FUNCTION_BLOCK FB_KF300 EXTENDS FB_Modbus_Tcp
(*
********************************************************************************
* Name: FB_KF300
*
* Author:  Automanh
* Version: 1.0.0
*
* Description:
*  KF300 Control for ShenChen
*
* Remarks:
*
* Revisions:
*   1.0 -AutomanH Rebuild
*********************************************************************************)
VAR_INPUT
	xIReset:BOOL;
	xIManualMode:BOOL;
	xIAutoMode:BOOL;
	xIEstop:BOOL;
	xIDeviceRunning:BOOL;
	LocalClient:stModbusPara;
	stRunPara	:ST_SetPara;//运行参数	
	stDeviceOpe	: stEasyPumpHmi;//操作按钮
END_VAR
VAR_OUTPUT
 	xQRdyCmd:BOOL;
	xQError:BOOL;
	xQBusy:BOOL;
	xQDone:BOOL;
	strQErrorID:STRING;
	xQCalibrationOK:BOOL;
	rMaxRunTime	:REAL;//最大运行时间,单位s
	rMinRunTime	:REAL;//最小运行时间,单位s
END_VAR
VAR
 	xStart:BOOL;
 {attribute 'tc_no_symbol'}
 iParaStep,iOldParaStep,iRunStep,iOldRunStep:INT;
 {attribute 'tc_no_symbol'}
 iCalibStep,iOldCalibStep:INT;
 {attribute 'tc_no_symbol'}
 stLocalPara:ST_LocalPara;
 {attribute 'tc_no_symbol'}
 stPara,stRun,stCalibInit,stCalibAction,stAdjust:ST_StepStatus; 
 {attribute 'tc_no_symbol'}
 stPump:st_EasyPump;
  {attribute 'tc_no_symbol'}
	tTimeout:ARRAY[1..5] OF TON;
 {attribute 'tc_no_symbol'}
	// 蠕动泵读取的液量
	rCurrVolum: REAL;
	{attribute 'tc_no_symbol'}
	//从蠕动泵读取的参数
	stReadPara:ST_ReadPara;
	{attribute 'tc_no_symbol'}
	// 数据数组
	arwData: ARRAY[1..2] OF WORD;
	{attribute 'tc_no_symbol'}
	eErrorID		: PumpError;(*错误码*)
	{attribute 'tc_no_symbol'}
	// 根据设定计算的转速
	rSetSpeed: REAL;
	{attribute 'tc_no_symbol'}
	// 设定的数据
	arwSetData: ARRAY [1..2] OF WORD;
	{attribute 'tc_no_symbol'}
	// 虚拟的较大时间
	rVirtualTime: REAL;
	{attribute 'tc_no_symbol'}
	OperR_TRIG:ARRAY[1..20] OF R_TRIG;
	{attribute 'tc_no_symbol'}
	// 循环计数
	i: INT;
	{attribute 'tc_no_symbol'}
	// 操作类型
	iOperType: INT;
	{attribute 'tc_no_symbol'}
	iOperCounter:INT;
	{attribute 'tc_no_symbol'}
	artDelay:ARRAY[1..5] OF TON;
	{attribute 'tc_no_symbol'}
	tSetTime:TIME;
	tModuleDelay:TON;
	iCalibNum:INT:=1;//校准灌装次数
END_VAR

MEMCPY(ADR(SUPER^.stModbusPara),ADR(LocalClient),SIZEOF(localClient));
SUPER^.M_Modbus();
ACT_RunPara();
ACT_Operation();
ACT_Running();
ACT_ParaCalc();
ACT_Calibration();
ACT_Reset();
ACT_Error();

ACTION ACT_Calibration:
CASE iCalibStep OF
 			0://等待启动
				 IF	stCalibInit.xStart THEN
							stCalibInit.xStart:=FALSE;
							stCalibInit.xBusy:=TRUE;
							stCalibInit.xDone:=FALSE;	
							iCalibStep:=10;//初始化校准参数
				 ELSIF stCalibAction.xStart THEN
						 	 stCalibAction.xStart :=FALSE;
							 stCalibAction.xBusy :=TRUE;
							 stCalibAction.xDone :=FALSE;
							 iCalibStep:=20;//校准
					ELSIF stAdjust.xStart THEN
					 		 stAdjust.xStart :=FALSE;
							 stAdjust.xBusy :=TRUE;
							 stAdjust.xDone :=FALSE;
							 iCalibStep:=30;//微调
				 END_IF
			10://初始化校准参数
					 iOldCalibStep:=iCalibStep;
					 arwDataWriteRegs[1]:=1;
					 wQuantityWriteRegs:=1;
					 wMBAddWriteRegs:=2007;
					 xWriteRegs:=TRUE;
					 IF  fbWriteRegs.bBusy THEN
							 xWriteRegs:=FALSE;
							 iCalibStep:=iCalibStep+1;
					END_IF
			11://液量设定完成
							 iOldCalibStep:=iCalibStep;
						 IF  NOT 	fbWriteRegs.bBusy AND  NOT  	fbWriteRegs.bError THEN
										iCalibStep:=iCalibStep+1;
							ELSIF   	fbReadRegs.bError THEN
									 iCalibStep:=999;				
									 eErrorID:=PumpError.FLT_SET_PARA;					
							END_IF		
		
			12://初始化校准参数完成
						 stCalibInit.xBusy:=FALSE;
							stCalibInit.xDone:=TRUE;	
						 	iCalibStep:=0;
						 
			
			 20://检查实际液量与设定液量的误差范围
					 IF   (stLocalPara.rFluVolumeSet - stLocalPara.iModuleRealVolume )<stLocalPara.rFluVolumeSet*0.5 THEN
							 //误差不能超过0.3ml
							 iCalibStep:=iCalibStep +1;				
					 ELSE
								 eERRORID := PumpError.FLT_Calib_OverFlow;//误差过大
								 iCalibStep:=999;	
					 END_IF
			 21://需要设定实际液量--实际液量最好是三组液量的平均值
							iOldCalibStep:=iCalibStep;
							MEMCPY(ADR(arwSetData[1]),ADR(stLocalPara.iModuleRealVolume),SIZEOF(stLocalPara.iModuleRealVolume) ); 
							arwDataWriteRegs[1]:=arwSetData[2];
							arwDataWriteRegs[2]:=arwSetData[1];
							wQuantityWriteRegs:=2;
							wMBAddWriteRegs:=2004;
							xWriteRegs:=TRUE;
							IF  fbWriteRegs.bBusy THEN
									xWriteRegs:=FALSE;
									 iCalibStep:=iCalibStep +1;		
						 END_IF
			 22://液量设定完成
							iOldCalibStep:=iCalibStep;
						 IF  NOT 	fbWriteRegs.bBusy AND  NOT  	fbWriteRegs.bError THEN
											 iCalibStep:=iCalibStep +1;		
							ELSIF   	fbReadRegs.bError THEN
										 iCalibStep:=999;				
										 eErrorID:=PumpError.FLT_CALIB_PARA;					
							END_IF		
			 23://校准实际液量设定结束
						 stCalibAction.xBusy :=FALSE;
						 stCalibAction.xDone :=TRUE;
						 iCalibStep:=0;				 
			30://校准微调-微调幅度为(设定量*0.001),这里要根据客户要求的精度进行调整
					 xQCalibrationOK:=FALSE;
					 iCalibStep:=iCalibStep +1;
			31://检测数据是否在精度范围内
					 iOldCalibStep:=iCalibStep;
					 IF  stLocalPara.iModuleRealVolume>=stLocalPara.rFluVolumeSet-(stLocalPara.rFluVolumeSet*stLocalPara.iAccuracySet) AND 
							 stLocalPara.iModuleRealVolume<=stLocalPara.rFluVolumeSet+(stLocalPara.rFluVolumeSet*stLocalPara.iAccuracySet) THEN
							 	 xQCalibrationOK:=TRUE;
								 iCalibStep:=36;
					ELSIF stLocalPara.iModuleRealVolume>=stLocalPara.rFluVolumeSet-(stLocalPara.rFluVolumeSet*stLocalPara.iAccuracySet) THEN
								 iCalibStep:=iCalibStep +1;	//需要减小
					ELSIF  stLocalPara.iModuleRealVolume<=stLocalPara.rFluVolumeSet+(stLocalPara.rFluVolumeSet*stLocalPara.iAccuracySet) THEN
								 iCalibStep:=iCalibStep +3;	//需要增大
					END_IF
			32://发送微调指令
					iOldParaStep:=iParaStep;
					arwDataWriteRegs[1]:=0;
					wQuantityWriteRegs:=1;
					wMBAddWriteRegs:=2006;
					xWriteRegs:=TRUE;
					IF  fbWriteRegs.bBusy THEN
							xWriteRegs:=FALSE;
							iCalibStep:=iCalibStep+1;
				 END_IF
		  33://微调执行完成
					 iOldParaStep:=iParaStep;
					 IF  NOT 	fbWriteRegs.bBusy AND  NOT  	fbWriteRegs.bError THEN
									 iCalibStep:=36;
						ELSIF   	fbReadRegs.bError THEN
								 iCalibStep:=999;				
								 eErrorID:=PumpError.FLT_SET_PARA;					
						END_IF			 
			34://发送微调指令
					iOldParaStep:=iParaStep;
					arwDataWriteRegs[1]:=1;
					wQuantityWriteRegs:=1;
					wMBAddWriteRegs:=2006;
					xWriteRegs:=TRUE;
					IF  fbWriteRegs.bBusy THEN
							xWriteRegs:=FALSE;
							iCalibStep:=iCalibStep+1;
				 END_IF
		  35://微调执行完成
					 iOldParaStep:=iParaStep;
					 IF  NOT 	fbWriteRegs.bBusy AND  NOT  	fbWriteRegs.bError THEN
									 iCalibStep:=36;
						ELSIF   	fbReadRegs.bError THEN
								 iCalibStep:=999;				
								 eErrorID:=PumpError.FLT_SET_PARA;					
						END_IF			 			
			 36://微调完成
							 stAdjust.xBusy :=FALSE;
							 stAdjust.xDone :=TRUE;
							 iCalibStep:=0;//校准			
END_CASE
 //防止程序二次执行
 IF	stCalibInit.xBusy THEN
			stCalibInit.xStart:=FALSE;
 ELSIF stCalibAction.xBusy THEN
			stCalibAction.xStart :=FALSE;
 ELSIF stAdjust.xBusy THEN
			stAdjust.xStart :=FALSE;
 END_IF
END_ACTION

ACTION ACT_Error:
tTimeout[1](IN:= iParaStep =iOldParaStep AND iParaStep<>0 , PT:= T#15S, Q=> , ET=> );
tTimeout[2](IN:= iRunStep =iOldRunStep AND iRunStep<>0 , PT:= T#15S, Q=> , ET=> );
tTimeout[3](IN:= iCalibStep =iOldCalibStep AND iCalibStep<>0 , PT:= T#15S, Q=> , ET=> );
IF		tTimeout[1].Q THEN
	  	stPara.xError:=TRUE;
	  	stPara.xBusy:=FALSE;
			eErrorID:=PumpError.FLT_CMD_TIMEOUT;
	    iParaStep := 999;
END_IF

IF		tTimeout[2].Q THEN
			stRun.xError:=TRUE;
			stRun.xBusy:=FALSE;
			eErrorID:=PumpError.FLT_CMD_TIMEOUT;
			iRunStep := 999;
END_IF

IF		tTimeout[3].Q THEN
			stAdjust.xError:=TRUE;
			stAdjust.xBusy:=FALSE;
			eErrorID:=PumpError.FLT_CMD_TIMEOUT;
			iCalibStep := 999;
END_IF

IF  eErrorID <> PumpError.NO_ERROR THEN
		xQError:=TRUE;
END_IF
//报错内容输出
CASE eErrorID OF 
		 PumpError.No_ERROR:
			 strQErrorID:='NO ERROR';
		 PumpError.FLT_PARA:
			 strQErrorID:='FLT_PARA';
		 PumpError.FLT_FLUVOLUM_TIME_PARA:
			 strQErrorID:='FLT_FLUVOLUM_TIME_PARA';
		 PumpError.FLT_SET_PARA:
			 strQErrorID:='FLT_SET_PARA';	
		 PumpError.FLT_CMD_TIMEOUT:
			 strQErrorID:='FLT_CMD_TIMEOUT';	
		 PumpError.FLT_RUN_ERROR:
			 strQErrorID:='FLT_RUN_ERROR';
		 PumpError.FLT_Calib_OverFlow:
			 strQErrorID:='FLT_Calib_OverFlow';	
		 PumpError.FLT_CALIB_PARA:
			 strQErrorID:='FLT_CALIB_PARA';		
		 PumpError.FLT_CONFIGURE_PARA:
			 strQErrorID:='FLT_CONFIGURE_PARA';		
END_CASE
END_ACTION

ACTION ACT_Operation:
OperR_TRIG[1](CLK:= (xIManualMode AND  stDeviceOpe.xPush_Hmi[1]) OR((xIAutoMode OR  xIDeviceRunning) AND stDeviceOpe.xPush_Auto[1]) , Q=> );	//Push
OperR_TRIG[2](CLK:= (xIManualMode AND  stDeviceOpe.xPush_Hmi[2]) OR((xIAutoMode OR  xIDeviceRunning) AND stDeviceOpe.xPush_Auto[2]) , Q=> );	//Push
OperR_TRIG[3](CLK:= (xIManualMode AND  stDeviceOpe.xPush_Hmi[3]) OR((xIAutoMode OR  xIDeviceRunning) AND stDeviceOpe.xPush_Auto[3]) , Q=> );	//Push
OperR_TRIG[4](CLK:= (xIManualMode AND  stDeviceOpe.xPush_Hmi[4]) OR((xIAutoMode OR  xIDeviceRunning) AND stDeviceOpe.xPush_Auto[4]) , Q=> );	//Push
OperR_TRIG[5](CLK:= (xIManualMode AND  stDeviceOpe.xPush_Hmi[5]) OR((xIAutoMode OR  xIDeviceRunning) AND stDeviceOpe.xPush_Auto[5]) , Q=> );	//Push
OperR_TRIG[6](CLK:= (xIManualMode AND  stDeviceOpe.xPull_Hmi[1]) OR((xIAutoMode OR  xIDeviceRunning) AND stDeviceOpe.xPull_Auto[1]) , Q=> );	//Pull
OperR_TRIG[7](CLK:= (xIManualMode AND  stDeviceOpe.xPull_Hmi[2]) OR((xIAutoMode OR  xIDeviceRunning) AND stDeviceOpe.xPull_Auto[2]) , Q=> );	//Pull
OperR_TRIG[8](CLK:= (xIManualMode AND  stDeviceOpe.xPull_Hmi[3]) OR((xIAutoMode OR  xIDeviceRunning) AND stDeviceOpe.xPull_Auto[3]) , Q=> );	//Pull
OperR_TRIG[9](CLK:= (xIManualMode AND  stDeviceOpe.xPull_Hmi[4]) OR((xIAutoMode OR  xIDeviceRunning) AND stDeviceOpe.xPull_Auto[4]) , Q=> );	//Pull
OperR_TRIG[10](CLK:= (xIManualMode AND  stDeviceOpe.xPull_Hmi[5]) OR((xIAutoMode OR  xIDeviceRunning) AND stDeviceOpe.xPull_Auto[5]) , Q=> );	//Pull
OperR_TRIG[11](CLK:= (xIManualMode AND  stDeviceOpe.xModulePush_Hmi) OR((xIAutoMode OR  xIDeviceRunning) AND stDeviceOpe.xModulePush_Auto) , Q=> );		//ModulePush	
OperR_TRIG[12](CLK:= (xIManualMode AND  stDeviceOpe.xFullSpeedPush_Hmi) OR((xIAutoMode OR  xIDeviceRunning) AND stDeviceOpe.xFullSpeedPush_Auto) , Q=> );//FullSpeedPush
OperR_TRIG[13](CLK:= (xIManualMode AND  stDeviceOpe.xFullSpeedPull_Hmi) OR((xIAutoMode OR  xIDeviceRunning) AND stDeviceOpe.xFullSpeedPull_Auto) , Q=> );//FullSpeedPull
OperR_TRIG[14](CLK:= (xIManualMode AND  stDeviceOpe.xFullSpeedStop_Hmi) OR((xIAutoMode OR  xIDeviceRunning) AND stDeviceOpe.xFullSpeedStop_Auto) , Q=> );//FullSpeedStop
OperR_TRIG[15](CLK:= (xIManualMode AND  stDeviceOpe.xStop_Hmi) OR((xIAutoMode OR  xIDeviceRunning) AND stDeviceOpe.xStop_Auto  ) , Q=> );//Stop
OperR_TRIG[16](CLK:= (xIManualMode AND  stDeviceOpe.xCalibAction_Hmi) OR((xIAutoMode OR  xIDeviceRunning) AND stDeviceOpe.xCalibAction_Auto) , Q=> );//Calibration Action
OperR_TRIG[17](CLK:= (xIManualMode AND  stDeviceOpe.xCalibInit_Hmi) OR((xIAutoMode OR  xIDeviceRunning) AND stDeviceOpe.xCalibInit_Auto), Q=> );//Calibration Init
OperR_TRIG[18](CLK:= (xIManualMode AND  stDeviceOpe.xAdjust_Hmi) OR((xIAutoMode OR  xIDeviceRunning) AND stDeviceOpe.xAdjust_Auto), Q=> );//Adjust
OperR_TRIG[19](CLK:= xIEstop, Q=> );//Estop

FOR  i:= 1 TO 20 BY 1 DO
 	IF   OperR_TRIG[i].Q THEN
				iOperCounter:= i;
				xStart:=TRUE;
				EXIT;
	END_IF
END_FOR
//Push
FOR  i:=1 TO 5 BY 1 DO
 		IF   iOperCounter =i THEN
		 		stLocalPara.rFluVolumeSet	:=stRunPara.rPushFluVolume[i];
				stLocalPara.rRuntimeSet	:=stRunPara.rPushRuntime[i];
				stLocalPara.iCycleNumber	:=stRunPara.iPushCycleNumber[i];
				stLocalPara.iBackAngle:=stRunPara.iPushBackAngle[i];
				stLocalPara.iDirectionSet:=stRunPara.iDirectionSet;
				stLocalPara.rVirualTime:=rMaxRunTime -1;
				iOperType:=stOperType.iPush;
		END_IF
END_FOR
//pull
FOR  i:=6 TO 10 BY 1 DO
 		IF   iOperCounter =i THEN
		 		stLocalPara.rFluVolumeSet	:=stRunPara.rPullFluVolume[i-5];
				stLocalPara.rRuntimeSet	:=stRunPara.rPullRuntime[i-5];
				stLocalPara.iCycleNumber	:=stRunPara.iPullCycleNumber[i-5];
				stLocalPara.iBackAngle:=stRunPara.iPullBackAngle[i-5];
				stLocalPara.iDirectionSet:=ABS(1-stRunPara.iDirectionSet);
				stLocalPara.rVirualTime:=rMaxRunTime -1;
				iOperType:=stOperType.iPull;
		END_IF
END_FOR 
 //Module Push
IF   iOperCounter =11 THEN
		 		stLocalPara.rFluVolumeSet	:=stRunPara.rCalFluVolume;
				stLocalPara.rRuntimeSet	 :=stRunPara.rCalTime;
				stLocalPara.iCycleNumber :=stRunPara.rCalNum;
				stLocalPara.iBackAngle:=stRunPara.rCalBackAngle;
				stLocalPara.iDirectionSet:=stRunPara.iDirectionSet;
				stLocalPara.iModuleAdress:=stRunPara.iModuleAdress;
				stLocalPara.iModuleSpeed:= stRunPara.rCalFluVolume * 60.0/(stRunPara.rSpeedRatio* stRunPara.rCalTime);
				stLocalPara.rVirualTime:=rMaxRunTime -1;
				iOperType:=stOperType.iModulePush;
////FullSpeedPush
ELSIF  iOperCounter =12 THEN
 				stLocalPara.iDirectionSet:=stRunPara.iDirectionSet;
 				iOperType:=stOperType.iFullSpeedPush;
ELSIF  iOperCounter =13 THEN
 			stLocalPara.iDirectionSet:=ABS(1-stRunPara.iDirectionSet);
 			iOperType:=stOperType.iFullSpeedPull;
ELSIF  iOperCounter =14 THEN
 			iOperType:=stOperType.iFullSpeedStop;
ELSIF  iOperCounter =15 OR iOperCounter =19  THEN
 			iOperType:=stOperType.iStop;
ELSIF  iOperCounter =16  THEN//Calibration
 			stLocalPara.iModuleRealVolume:=stRunPara.rModuleRealFluVolume;
 			iOperType:=stOperType.iCalibAction;
ELSIF  iOperCounter =17  THEN
 			iOperType:=stOperType.iCalibInit;	
ELSIF    iOperCounter =18 THEN //adjust
 			stLocalPara.iModuleRealVolume:=stRunPara.rModuleRealFluVolume;
 			stLocalPara.iAccuracySet:=stRunPara.iAccuracySet;
 			iOperType:=stOperType.iAdjust;	
END_IF


MEMSET(ADR(stDeviceOpe),0,SIZEOF(stDeviceOpe));
END_ACTION

ACTION ACT_ParaCalc:
//
(*************************检测配置参数是否匹配成功*********************************)
IF stRunPara.iPumpType=RudongPump_PumpType.DFPluse THEN
	//MiniPump泵头
	IF  stRunPara.iPumpTypeSet=RudongPump_PumpHeadType.MiniPump01 THEN
		stPump.iPumpType:=0;//泵头值为0
			IF stRunPara.iHosePipeTypeSet=RudongPump_SoftPipeType.P13 THEN//13#软管
				stPump.iHosePipeType:=13;//软管类型值13
				IF  stLocalPara.rFluVolumeSet*1000/135<0.1 THEN
					rMaxRunTime:=	0.1;
				ELSE
					rMaxRunTime:=	stLocalPara.rFluVolumeSet*1000/135;
				END_IF
				rMaxRunTime:=	(stLocalPara.rFluVolumeSet/0.45)*0.2;//最大流量(0.45微升/秒,0.0024ml/min)	
			ELSIF stRunPara.iHosePipeTypeSet=RudongPump_SoftPipeType.P14 THEN//14#软管
					stPump.iHosePipeType:=13;//软管类型值13
				IF stLocalPara.rFluVolumeSet*1000/570<0.1 THEN
							rMinRunTime:=	0.1;
				ELSE
						rMinRunTime:=	stLocalPara.rFluVolumeSet*1000/135;
				END_IF
				rMaxRunTime:=	(stLocalPara.rFluVolumeSet/1.9)*0.2;	
			ELSIF stRunPara.iHosePipeTypeSet=RudongPump_SoftPipeType.P19 THEN//19#软管
				stPump.iHosePipeType:=19;
				IF stLocalPara.rFluVolumeSet*1000/1240<0.1 THEN
					rMinRunTime:=	0.1;
				ELSE
					rMinRunTime:=	stLocalPara.rFluVolumeSet*1000/1240;
				END_IF
					rMaxRunTime:=	(stLocalPara.rFluVolumeSet*1000/4.13)*0.2;		
			ELSIF stRunPara.iHosePipeTypeSet=RudongPump_SoftPipeType.P16 THEN//16#软管
					stPump.iHosePipeType:=16;
				IF stLocalPara.rFluVolumeSet*1000/1880<0.1 THEN
					rMinRunTime:=	0.1;
				ELSE
					rMinRunTime:=	stLocalPara.rFluVolumeSet*1000/1880;
				END_IF
				rMaxRunTime:=	(stLocalPara.rFluVolumeSet*1000/6.28)*0.2;	
			ELSIF stRunPara.iHosePipeTypeSet=RudongPump_SoftPipeType.P25 THEN//25#软管
					stPump.iHosePipeType:=25;
				IF stLocalPara.rFluVolumeSet*1000/3100<0.1 THEN
					rMinRunTime:=	0.1;
				ELSE
					rMinRunTime:=	stLocalPara.rFluVolumeSet*1000/3100;
				END_IF
				rMaxRunTime:=	(stLocalPara.rFluVolumeSet*1000/10.33)*0.2;			
		ELSE
				eERRORID:=RudongPump_ERROR.FLT_CONFIGURE_PARA;		
		END_IF
	//UD15
	ELSIF  stRunPara.iPumpTypeSet=RudongPump_PumpHeadType.UD15 THEN
				stPump.iHosePipeType:=1;//泵头值为0
			IF stRunPara.iHosePipeTypeSet=RudongPump_SoftPipeType.P16 THEN//16#软管
				stPump.iHosePipeType:=16;
				IF stLocalPara.rFluVolumeSet*1000/4000<0.1 THEN
					rMinRunTime:=	0.1;
				ELSE
					rMinRunTime:=	stLocalPara.rFluVolumeSet*1000/4000;
				END_IF
				rMaxRunTime:=	(stLocalPara.rFluVolumeSet*1000/13.33)*0.2;		
			ELSIF stRunPara.iHosePipeTypeSet=RudongPump_SoftPipeType.P17 THEN//17#软管
				stPump.iHosePipeType:=17;
				IF stLocalPara.rFluVolumeSet*1000/15000<0.1 THEN
					rMinRunTime:=	0.1;
				ELSE
					rMinRunTime:=	stLocalPara.rFluVolumeSet*1000/15000;
				END_IF
				rMaxRunTime:=	(stLocalPara.rFluVolumeSet*1000/50)*0.2;	
			ELSIF stRunPara.iHosePipeTypeSet=RudongPump_SoftPipeType.P25 THEN//25#软管
				stPump.iHosePipeType:=25;
				IF stLocalPara.rFluVolumeSet*1000/8000<0.1 THEN
					rMinRunTime:=	0.1;
				ELSE
					rMinRunTime:=	stLocalPara.rFluVolumeSet*1000/8000;
				END_IF
				 rMaxRunTime:=	(stLocalPara.rFluVolumeSet*1000/26.66)*0.2;			
		ELSE
				eERRORID:=RudongPump_ERROR.FLT_CONFIGURE_PARA;		
		END_IF
	//HandyPump01泵头
ELSIF  stRunPara.iPumpTypeSet=RudongPump_PumpHeadType.HandyPump01 THEN
 			IF stRunPara.iHosePipeTypeSet=RudongPump_SoftPipeType.P13 THEN//13#软管,三滚轮
				IF stLocalPara.rFluVolumeSet*1000/155<0.1 THEN
					rMinRunTime:=	0.1;
				ELSE
					rMinRunTime:=	stLocalPara.rFluVolumeSet*1000/155;
				END_IF
					rMaxRunTime:=	(stLocalPara.rFluVolumeSet*1000/0.51)*0.2;	
		
	(*	IF stRunPara.iHosePipeTypeSet=RudongPump_SoftPipeType.P13 THEN//13#软管,三滚轮
			iMinRunTime:=	(rFluVolumeSet/10)*60;
			iMaxRunTime:=	(rFluVolumeSet/0.0033)*60;	
		ELSIF stRunPara.iHosePipeTypeSet=RudongPump_SoftPipeType.P14 THEN//14#软管,三滚轮
			iMinRunTime:=	(rFluVolumeSet/56)*60;
			iMaxRunTime:=	(rFluVolumeSet/0.0187)*60;		
		ELSIF stRunPara.iHosePipeTypeSet=RudongPump_SoftPipeType.P19 THEN//19#软管,三滚轮
			iMinRunTime:=	(rFluVolumeSet/111)*60;
			iMaxRunTime:=	(rFluVolumeSet/0.0371)*60;
		ELSIF stRunPara.iHosePipeTypeSet=RudongPump_SoftPipeType.P16 THEN//16#软管,三滚轮
			iMinRunTime:=	(rFluVolumeSet/190)*60;
			iMaxRunTime:=	(rFluVolumeSet/0.0636)*60;		
		ELSIF stRunPara.iHosePipeTypeSet=RudongPump_SoftPipeType.P25 THEN//25#软管,三滚轮
			iMinRunTime:=	(rFluVolumeSet/365)*60;
			iMaxRunTime:=	(rFluVolumeSet/0.1219)*60;
	*)
		ELSE
				eERRORID:=RudongPump_ERROR.FLT_CONFIGURE_PARA;						
		END_IF
	END_IF
ELSE
		eERRORID:=RudongPump_ERROR.FLT_CONFIGURE_PARA;
END_IF


(*
//MiniPump01泵头
IF  stRunPara.iPumpTypeSet=RudongPump_PumpHeadType.MiniPump01 THEN
		IF stRunPara.iHosePipeTypeSet=RudongPump_SoftPipeType.P13 THEN//13#软管
			iMinRunTime:=	(rFluVolumeSet/8)*60;//最大流量(135微升/秒,8.28ml/min)
			iMaxRunTime:=	(rFluVolumeSet/0.45)*60;//最大流量(0.45微升/秒,0.0024ml/min)	
		ELSIF stRunPara.iHosePipeTypeSet=RudongPump_SoftPipeType.P14 THEN//14#软管
			iMinRunTime:=	(rFluVolumeSet/33)*60;
			iMaxRunTime:=	(rFluVolumeSet/1.9)*60;
		ELSIF stRunPara.iHosePipeTypeSet=RudongPump_SoftPipeType.P19 THEN//19#软管
			iMinRunTime:=	(rFluVolumeSet/77)*60;
			iMaxRunTime:=	(rFluVolumeSet/4.13)*60;	
		ELSIF stRunPara.iHosePipeTypeSet=RudongPump_SoftPipeType.P16 THEN//16#软管
			iMinRunTime:=	(rFluVolumeSet/114)*60;
			iMaxRunTime:=	(rFluVolumeSet/6.28)*60;	
		ELSIF stRunPara.iHosePipeTypeSet=RudongPump_SoftPipeType.P25 THEN//25#软管
			iMinRunTime:=	(rFluVolumeSet/190)*60;
			iMaxRunTime:=	(rFluVolumeSet/10.33)*60;		
		ELSIF stRunPara.iHosePipeTypeSet=RudongPump_SoftPipeType.P1_1 THEN//1x1#软管
			iMinRunTime:=	(rFluVolumeSet/15)*60;
			iMaxRunTime:=	(rFluVolumeSet/4.5)*60;	
		ELSIF stRunPara.iHosePipeTypeSet=RudongPump_SoftPipeType.P2_1 THEN//2x1#软管
			iMinRunTime:=	(rFluVolumeSet/54)*60;
			iMaxRunTime:=	(rFluVolumeSet/4.5)*60;		
		ELSIF stRunPara.iHosePipeTypeSet=RudongPump_SoftPipeType.P2_5_1 THEN//2.5x1#软管
			iMinRunTime:=	(rFluVolumeSet/76)*60;
			iMaxRunTime:=	(rFluVolumeSet/5)*60;		
		ELSIF stRunPara.iHosePipeTypeSet=RudongPump_SoftPipeType.P3_1 THEN//3x1#软管
			iMinRunTime:=	(rFluVolumeSet/108)*60;
			iMaxRunTime:=	(rFluVolumeSet/5)*60;
	ELSE
			eERRORID:=RudongPump_ERROR.FLT_CONFIGURE_PARA;		
	END_IF		
	
//MiniPump02泵头
ELSIF  stRunPara.iPumpTypeSet=RudongPump_PumpHeadType.MiniPump02 THEN
	IF stRunPara.iHosePipeTypeSet=RudongPump_SoftPipeType.P1_1 THEN//1x1#软管
		iMinRunTime:=	(rFluVolumeSet/15.01)*60;
		iMaxRunTime:=	(rFluVolumeSet/0.005)*60;	
	ELSIF stRunPara.iHosePipeTypeSet=RudongPump_SoftPipeType.P2_1 THEN//2x1#软管
		iMinRunTime:=	(rFluVolumeSet/54.63)*60;
		iMaxRunTime:=	(rFluVolumeSet/0.018)*60;		
	ELSIF stRunPara.iHosePipeTypeSet=RudongPump_SoftPipeType.P2_5_1 THEN//2.5x1#软管
		iMinRunTime:=	(rFluVolumeSet/76.84)*60;
		iMaxRunTime:=	(rFluVolumeSet/0.0256)*60;
	ELSE
			eERRORID:=RudongPump_ERROR.FLT_CONFIGURE_PARA;						
	END_IF	

//HandyPump01泵头
ELSIF  stRunPara.iPumpTypeSet=RudongPump_PumpHeadType.HandyPump01 THEN
	IF stRunPara.iHosePipeTypeSet=RudongPump_SoftPipeType.P13 THEN//13#软管,三滚轮
		iMinRunTime:=	(rFluVolumeSet/10)*60;
		iMaxRunTime:=	(rFluVolumeSet/0.0033)*60;	
	ELSIF stRunPara.iHosePipeTypeSet=RudongPump_SoftPipeType.P14 THEN//14#软管,三滚轮
		iMinRunTime:=	(rFluVolumeSet/56)*60;
		iMaxRunTime:=	(rFluVolumeSet/0.0187)*60;		
	ELSIF stRunPara.iHosePipeTypeSet=RudongPump_SoftPipeType.P19 THEN//19#软管,三滚轮
		iMinRunTime:=	(rFluVolumeSet/111)*60;
		iMaxRunTime:=	(rFluVolumeSet/0.0371)*60;
	ELSIF stRunPara.iHosePipeTypeSet=RudongPump_SoftPipeType.P16 THEN//16#软管,三滚轮
		iMinRunTime:=	(rFluVolumeSet/190)*60;
		iMaxRunTime:=	(rFluVolumeSet/0.0636)*60;		
	ELSIF stRunPara.iHosePipeTypeSet=RudongPump_SoftPipeType.P25 THEN//25#软管,三滚轮
		iMinRunTime:=	(rFluVolumeSet/365)*60;
		iMaxRunTime:=	(rFluVolumeSet/0.1219)*60;
	ELSE
			eERRORID:=RudongPump_ERROR.FLT_CONFIGURE_PARA;						
	END_IF

//HandyPump02泵头
ELSIF  stRunPara.iPumpTypeSet=RudongPump_PumpHeadType.HandyPump02 THEN
	IF stRunPara.iHosePipeTypeSet=RudongPump_SoftPipeType.P13 THEN//13#软管,三滚轮
		iMinRunTime:=	(rFluVolumeSet/10)*60;
		iMaxRunTime:=	(rFluVolumeSet/0.0033)*60;	
	ELSIF stRunPara.iHosePipeTypeSet=RudongPump_SoftPipeType.P14 THEN//14#软管,三滚轮
		iMinRunTime:=	(rFluVolumeSet/56)*60;
		iMaxRunTime:=	(rFluVolumeSet/0.0187)*60;		
	ELSIF stRunPara.iHosePipeTypeSet=RudongPump_SoftPipeType.P19 THEN//19#软管,三滚轮
		iMinRunTime:=	(rFluVolumeSet/111)*60;
		iMaxRunTime:=	(rFluVolumeSet/0.0371)*60;
	ELSIF stRunPara.iHosePipeTypeSet=RudongPump_SoftPipeType.P16 THEN//16#软管,三滚轮
		iMinRunTime:=	(rFluVolumeSet/190)*60;
		iMaxRunTime:=	(rFluVolumeSet/0.0636)*60;	
	ELSE
			eERRORID:=RudongPump_ERROR.FLT_CONFIGURE_PARA;							
	END_IF

//EasyPumpI_III泵头,单通道
ELSIF  stRunPara.iPumpTypeSet=RudongPump_PumpHeadType.EasyPumpI_III THEN
	IF stRunPara.iHosePipeTypeSet=RudongPump_SoftPipeType.P13 THEN//13#软管
		iMinRunTime:=	(rFluVolumeSet/32)*60;
		iMaxRunTime:=	(rFluVolumeSet/0.0053)*60;	
	ELSIF stRunPara.iHosePipeTypeSet=RudongPump_SoftPipeType.P14 THEN//14#软管
		iMinRunTime:=	(rFluVolumeSet/162)*60;
		iMaxRunTime:=	(rFluVolumeSet/0.027)*60;		
	ELSIF stRunPara.iHosePipeTypeSet=RudongPump_SoftPipeType.P19 THEN//19#软管
		iMinRunTime:=	(rFluVolumeSet/330)*60;
		iMaxRunTime:=	(rFluVolumeSet/0.055)*60;
	ELSIF stRunPara.iHosePipeTypeSet=RudongPump_SoftPipeType.P16 THEN//16#软管
		iMinRunTime:=	(rFluVolumeSet/560)*60;
		iMaxRunTime:=	(rFluVolumeSet/0.093)*60;	
	ELSIF stRunPara.iHosePipeTypeSet=RudongPump_SoftPipeType.P25 THEN//25#软管
		iMinRunTime:=	(rFluVolumeSet/1180)*60;
		iMaxRunTime:=	(rFluVolumeSet/0.197)*60;	
	ELSIF stRunPara.iHosePipeTypeSet=RudongPump_SoftPipeType.P17 THEN//17#软管
		iMinRunTime:=	(rFluVolumeSet/2000)*60;
		iMaxRunTime:=	(rFluVolumeSet/0.333)*60;	
	ELSIF stRunPara.iHosePipeTypeSet=RudongPump_SoftPipeType.P18 THEN//18#软管
		iMinRunTime:=	(rFluVolumeSet/2580)*60;
		iMaxRunTime:=	(rFluVolumeSet/0.430)*60;	
	ELSE
			eERRORID:=RudongPump_ERROR.FLT_CONFIGURE_PARA;							
	END_IF

//EasyPumpII_IV泵头,单通道
ELSIF  stRunPara.iPumpTypeSet=RudongPump_PumpHeadType.EasyPumpII_IV THEN
	IF stRunPara.iHosePipeTypeSet=RudongPump_SoftPipeType.P15 THEN//15#软管
		iMinRunTime:=	(rFluVolumeSet/1080)*60;
		iMaxRunTime:=	(rFluVolumeSet/0.0180)*60;	
	ELSIF stRunPara.iHosePipeTypeSet=RudongPump_SoftPipeType.P24 THEN//24#软管
		iMinRunTime:=	(rFluVolumeSet/1640)*60;
		iMaxRunTime:=	(rFluVolumeSet/0.273)*60;		
	ELSIF stRunPara.iHosePipeTypeSet=RudongPump_SoftPipeType.P35 THEN//35#软管
		iMinRunTime:=	(rFluVolumeSet/2300)*60;
		iMaxRunTime:=	(rFluVolumeSet/0.383)*60;
	ELSIF stRunPara.iHosePipeTypeSet=RudongPump_SoftPipeType.P36 THEN//36#软管
		iMinRunTime:=	(rFluVolumeSet/3100)*60;
		iMaxRunTime:=	(rFluVolumeSet/0.517)*60;	
	ELSE
			eERRORID:=RudongPump_ERROR.FLT_CONFIGURE_PARA;							
	END_IF

//EasyPumpV_VI泵头,双通道
ELSIF  stRunPara.iPumpTypeSet=RudongPump_PumpHeadType.EasyPumpV_VI THEN
		IF stRunPara.iHosePipeTypeSet=RudongPump_SoftPipeType.P13 THEN//13#软管
		iMinRunTime:=	(rFluVolumeSet/32)*60;
		iMaxRunTime:=	(rFluVolumeSet/0.0053)*60;	
	ELSIF stRunPara.iHosePipeTypeSet=RudongPump_SoftPipeType.P14 THEN//14#软管
		iMinRunTime:=	(rFluVolumeSet/162)*60;
		iMaxRunTime:=	(rFluVolumeSet/0.0027)*60;		
	ELSIF stRunPara.iHosePipeTypeSet=RudongPump_SoftPipeType.P19 THEN//19#软管
		iMinRunTime:=	(rFluVolumeSet/330)*60;
		iMaxRunTime:=	(rFluVolumeSet/0.0055)*60;
	ELSIF stRunPara.iHosePipeTypeSet=RudongPump_SoftPipeType.P16 THEN//16#软管
		iMinRunTime:=	(rFluVolumeSet/560)*60;
		iMaxRunTime:=	(rFluVolumeSet/0.093)*60;		
	ELSIF stRunPara.iHosePipeTypeSet=RudongPump_SoftPipeType.P25 THEN//25#软管
		iMinRunTime:=	(rFluVolumeSet/1180)*60;
		iMaxRunTime:=	(rFluVolumeSet/0.197)*60;
	ELSE
			eERRORID:=RudongPump_ERROR.FLT_CONFIGURE_PARA;							
	END_IF
	
END_IF


END_IF

*)
		


//参数超出范围报错	
IF stLocalPara.rFluVolumeSet<>0 THEN
	IF stLocalPara.rRuntimeSet<rMinRunTime OR stLocalPara.rRuntimeSet>rMaxRunTime OR  rMaxRunTime<rMinRunTime THEN
		eERRORID:=RudongPump_ERROR.FLT_CONFIGURE_PARA;
	END_IF
END_IF
END_ACTION

ACTION ACT_Reset:
IF   xIReset THEN
 
 	 iParaStep:=0;
	 iRunStep:=0;
 	 iCalibStep:=0;
	 
	 iOldParaStep:=0;
	 iOldRunStep:=0;
	 iOldCalibStep:=0;
	 
	 stPara.xStart:=FALSE;
	 stPara.xBusy:=FALSE;
	 stPara.xError:=FALSE;
 
	 stRun.xStart:=FALSE;
	 stRun.xBusy:=FALSE;
	 stRun.xError:=FALSE;
		
	 stCalibInit.xStart:=FALSE;
	 stCalibInit.xBusy:=FALSE;
	 stCalibInit.xDone:=FALSE;
	 
	 stCalibAction.xStart:=FALSE;
	 stCalibAction.xBusy :=FALSE;
	 stCalibAction.xDone :=FALSE;
	 
	 stAdjust.xStart:=FALSE;
	 stAdjust.xBusy :=FALSE;
	 stAdjust.xDone :=FALSE;
	 
	
	 
	 xQBusy:=FALSE;
	 //xQDone:=FALSE;
	 
	 eErrorID := PumpError.NO_ERROR;
	 xIReset:=FALSE;
END_IF
END_ACTION

ACTION ACT_Running:
IF  NOT  xQBusy THEN
 		xQRdyCmd:=TRUE;
ELSE
 		xQRdyCmd:=FALSE;	
END_IF

CASE  iRunStep OF 
 0://等待开始
 		IF  xStart THEN
		 		xStart:=FALSE;
				xQBusy:=TRUE;
				xQDone:=FALSE;
				iRunStep:=iRunStep +1;
		END_IF
 1://检查是否是全速
 		IF    iOperType=stOperType.iFullSpeedPull OR 
					iOperType=stOperType.iFullSpeedPush OR
					iOperType=stOperType.iStop OR
					iOperType=stOperType.iFullSpeedStop THEN
					iRunStep:=iRunStep +3;
		ELSE
		 			iRunStep:=iRunStep +1;
 		END_IF
 2://参数传递
 		 iOldRunStep:=iRunStep;
 		 stPara.xStart:=TRUE;
		 IF   stPara.xBusy THEN
				 iRunStep:=iRunStep +1;
		 END_IF
 3://等待参数传递完成
 		 	iOldRunStep:=iRunStep;
 		 IF  stPara.xDone   THEN
				iRunStep:=iRunStep +1;
		 END_IF
 4://开始执行
 			iOldRunStep:=iRunStep;
	  IF 		 iOperType=stOperType.iPush OR
					 iOperType=stOperType.iPull  THEN
    				iRunStep:=10;
		ELSIF   iOperType=stOperType.iStop OR 
						iOperType=stOperType.iFullSpeedStop  THEN
    			  iRunStep:=20;
		ELSIF   iOperType=stOperType.iFullSpeedPull OR 
						iOperType=stOperType.iFullSpeedPush  THEN
		 				iRunStep:=30;
		ELSIF     iOperType=stOperType.iModulePush THEN
    				iRunStep:=40;
		ELSIF     iOperType=stOperType.iCalibAction THEN
    				iRunStep:=50;
		ELSIF  		iOperType=stOperType.iCalibInit THEN
		 				iRunStep:=60;
		ELSIF   		iOperType=stOperType.iAdjust THEN
		 				iRunStep:=70;
		END_IF	
 10://Pull/push
				iOldRunStep:=iRunStep;
				arwDataWriteRegs[1]:=1;//启动
				wQuantityWriteRegs:=1;
				wMBAddWriteRegs:=1011;
				xWriteRegs:=TRUE;
				IF  fbWriteRegs.bBusy THEN
						xWriteRegs:=FALSE;
						iRunStep:=iRunStep+1;
			 END_IF
 11://启动完成
			iOldRunStep:=iRunStep;
	  	IF  NOT 	fbWriteRegs.bBusy AND  NOT  	fbWriteRegs.bError THEN
	  	 				iRunStep:=iRunStep +1;
	  	 ELSIF   	fbWriteRegs.bError THEN
	  	 			iRunStep:=999;				
	  	 			eErrorID:=PumpError.FLT_RUN_ERROR;					
	  	 END_IF		
  12://等待运行结束
			iOldParaStep:=iParaStep;
			wMBAddReadRegs:=1011;
			wQuantityReadRegs:=1;
			xReadRegs:=TRUE;
			IF  fbReadRegs.bBusy THEN
			 	xReadRegs:=FALSE;
				iRunStep:=iRunStep+1;
			END_IF
	13://等待读取完成
			 	iOldParaStep:=iParaStep;
	  	  IF  NOT 	fbReadRegs.bBusy AND  NOT  	fbReadRegs.bError THEN
				 				 stReadPara.iRunning:=arwDataReadRegs[1];
	  		 				 iRunStep:=iRunStep+1;
	  		 ELSIF   	fbReadRegs.bError THEN
	  		 			iRunStep:=999;				
	  		 			eErrorID:=PumpError.FLT_READ_PARA;					
	  		 END_IF	
				 artDelay[1](IN:=FALSE);
	14://检查是否已经停止运行
				IF  stReadPara.iRunning =0 THEN
				 			iRunStep:=100;
				ELSE //再次读取
						artDelay[1](IN:= TRUE, PT:= T#100MS, Q=> , ET=> );
						IF  artDelay[1].Q  THEN
								 iRunStep:=12;
								 artDelay[1](IN:= FALSE);
						END_IF
				END_IF			 
	20://Stop
				 iOldRunStep:=iRunStep;
				 arwDataWriteRegs[1]:=0;//停止
				 arwDataWriteRegs[2]:=0;//全速停止
				 wQuantityWriteRegs:=2;
				 wMBAddWriteRegs:=1011;
				 xWriteRegs:=TRUE;
				 IF  fbWriteRegs.bBusy THEN
						 xWriteRegs:=FALSE;
						 iRunStep:=iRunStep+1;
				END_IF
	21://运行完成
			 iOldRunStep:=iRunStep;
			 IF  NOT 	fbWriteRegs.bBusy AND  NOT  	fbWriteRegs.bError THEN
							 iRunStep:=100;
				ELSIF   	fbWriteRegs.bError THEN
						 iRunStep:=999;				
						 eErrorID:=PumpError.FLT_RUN_ERROR;					
				END_IF				
	30://写入方向
				iOldParaStep:=iParaStep;
				MEMCPY(ADR(arwDataWriteRegs[1]),ADR(stLocalPara.iDirectionSet),SIZEOF (stLocalPara.iDirectionSet));
				wQuantityWriteRegs:=1;
				wMBAddWriteRegs:=1010;
				xWriteRegs:=TRUE;
				IF  fbWriteRegs.bBusy THEN
						xWriteRegs:=FALSE;
						iRunStep:=iRunStep+1;
			 END_IF
	 31://方向写入完成
			 iOldParaStep:=iParaStep;
			 IF  NOT 	fbWriteRegs.bBusy AND  NOT  	fbWriteRegs.bError THEN
							 iRunStep:=iRunStep +1;
				ELSIF   	fbWriteRegs.bError THEN
						 iRunStep:=999;				
						 eErrorID:=PumpError.FLT_SET_PARA;					
				END_IF		
	32://FullSpeed
				 iOldRunStep:=iRunStep;
				 arwDataWriteRegs[1]:=1;//全速启动
				 wQuantityWriteRegs:=1;
				 wMBAddWriteRegs:=1012;
				 xWriteRegs:=TRUE;
				 IF  fbWriteRegs.bBusy THEN
						 xWriteRegs:=FALSE;
						 iRunStep:=iRunStep+1;
				END_IF
	33://全速启动
			 iOldRunStep:=iRunStep;
			 IF  NOT 	fbWriteRegs.bBusy AND  NOT fbWriteRegs.bError THEN
							 iRunStep:=100;
				ELSIF   	fbWriteRegs.bError THEN
						 iRunStep:=999;				
						 eErrorID:=PumpError.FLT_RUN_ERROR;					
				END_IF	
	40://
			iCalibNum:=1;
			iRunStep:=iRunStep+1;
	41://Module Push
				 iOldRunStep:=iRunStep;
				 arwDataWriteRegs[1]:=1;//单元启动
				 wQuantityWriteRegs:=1;
				 wMBAddWriteRegs:=2003;
				 xWriteRegs:=TRUE;
				 IF  fbWriteRegs.bBusy THEN
						 xWriteRegs:=FALSE;
						 iRunStep:=iRunStep+1;
				END_IF
	42://单元启动注液
			 iOldRunStep:=iRunStep;
			 IF  NOT 	fbWriteRegs.bBusy AND  NOT fbWriteRegs.bError THEN
							 iRunStep:=iRunStep +1;
				ELSIF   	fbWriteRegs.bError THEN
						 iRunStep:=999;				
						 eErrorID:=PumpError.FLT_RUN_ERROR;					
				END_IF
	43://等待运行结束
			 iOldParaStep:=iParaStep;
			 wMBAddReadRegs:=2003;
			 wQuantityReadRegs:=1;
			 xReadRegs:=TRUE;
			 IF  fbReadRegs.bBusy THEN
				 xReadRegs:=FALSE;
				 iRunStep:=iRunStep+1;
			 END_IF
	 44://等待读取完成
				 iOldParaStep:=iParaStep;
				 IF  NOT 	fbReadRegs.bBusy AND  NOT  	fbReadRegs.bError THEN
									stReadPara.iRunning:=arwDataReadRegs[1];
									iRunStep:=iRunStep+1;
					ELSIF   	fbReadRegs.bError THEN
							 iRunStep:=999;				
							 eErrorID:=PumpError.FLT_READ_PARA;					
					END_IF	
					artDelay[1](IN:=FALSE);
	 45://检查是否已经停止运行
				 IF  stReadPara.iRunning =0 THEN
							 	iRunStep:=iRunStep +1;
				 ELSE //再次读取
						 artDelay[1](IN:= TRUE, PT:= T#100MS, Q=> , ET=> );
						 IF  artDelay[1].Q  THEN
									iRunStep:=12;
									artDelay[1](IN:= FALSE);
						 END_IF
				 END_IF		
		46://检查灌装次数
				iCalibNum:=iCalibNum +1 ;
				iRunStep:=iRunStep +1;
	  47://
				IF  iCalibNum > stLocalPara.iCycleNumber THEN
				 				iRunStep:=100;
				ELSE
								iRunStep:=iRunStep +1;		
				END_IF			 			 
		48://检查单元注液时间等待0.5
			 tModuleDelay(IN:=TRUE, PT:= T#1500MS, Q=> , ET=> );
			 IF	  	tModuleDelay.Q THEN
							 tModuleDelay(IN:=FALSE);	
							 iRunStep:=41;
			 END_IF	
			 
		50://写入实际液量	
					 MEMCPY(ADR(arwSetData[1]),ADR(stLocalPara.iModuleRealVolume),SIZEOF(stLocalPara.iModuleRealVolume) ); 
					 arwDataWriteRegs[1]:=arwSetData[2];
					 arwDataWriteRegs[2]:=arwSetData[1];
					 iRunStep:=iRunStep +1;
		
		51://开始写入
					 iOldRunStep:=iRunStep;
					 wQuantityWriteRegs:=2;
					 wMBAddWriteRegs:=2004;
					 xWriteRegs:=TRUE;
					 IF  fbWriteRegs.bBusy THEN
							 xWriteRegs:=FALSE;
							 iRunStep:=iRunStep+1;
					END_IF
		52://等待运行结束
				 iOldParaStep:=iParaStep;
				 wMBAddReadRegs:=1011;
				 wQuantityReadRegs:=1;
				 xReadRegs:=TRUE;
				 IF  fbReadRegs.bBusy THEN
					 xReadRegs:=FALSE;
					 iRunStep:=iRunStep+1;
				 END_IF
		 53://等待读取完成
					 iOldParaStep:=iParaStep;
					 IF  NOT 	fbReadRegs.bBusy AND  NOT  	fbReadRegs.bError THEN
										stReadPara.iRunning:=arwDataReadRegs[1];
										iRunStep:=iRunStep+1;
						ELSIF   	fbReadRegs.bError THEN
								 iRunStep:=999;				
								 eErrorID:=PumpError.FLT_READ_PARA;					
						END_IF	
						artDelay[1](IN:=FALSE);
		 54://检查是否已经停止运行
					 IF  stReadPara.iRunning =0 THEN
								 iRunStep:=100;
					 ELSE //再次读取
							 artDelay[1](IN:= TRUE, PT:= T#100MS, Q=> , ET=> );
							 IF  artDelay[1].Q  THEN
										iRunStep:=12;
										artDelay[1](IN:= FALSE);
							 END_IF
					 END_IF			 
		 60://初始化校准参数
					 stCalibInit.xStart :=TRUE;
					 iRunStep:=iRunStep +1;
		 61://等待
				 IF  stCalibInit.xBusy THEN
						 iRunStep:=iRunStep +1;
				 END_IF
		 62://完成
				 IF stCalibInit.xDone THEN
							 iRunStep:=100;
				 END_IF 
		 70://微调
					 stAdjust.xStart :=TRUE;
					 iRunStep:=iRunStep +1;
		 71://等待
				 IF  stAdjust.xBusy THEN
						 iRunStep:=iRunStep +1;
				 END_IF
		 72://完成
				 IF stAdjust.xDone THEN
							 iRunStep:=100;
				 END_IF 
	   100://等待S钟 
					artDelay[2](IN:=TRUE , PT:= T#1S, Q=> , ET=> );		 
					IF  artDelay[2].Q THEN
					     iRunStep:=iRunStep +1;
							 artDelay[2](IN:=FALSE);
					END_IF
		 101://运行结束
					xQBusy:=FALSE;
					xQDone:=TRUE;
					iRunStep:=0;
 END_CASE
 //防止程序二次执行
	IF  xQBusy THEN
		 		xStart:=FALSE;
  END_IF
END_ACTION

ACTION ACT_RunPara:
CASE iParaStep OF	
	0://开始
			IF   stPara.xStart THEN
			 		 stPara.xStart:=FALSE;
					 stPara.xBusy:=TRUE;
					 stPara.xDone:=FALSE;
					  iParaStep := iParaStep + 1;
			 END_IF
 	1://查流量设定的转速是否在0.1rpm-600rpm之间
			iOldParaStep:=iParaStep;
			IF 	stLocalPara.rRuntimeSet = 0  THEN 
					 eERRORID := PumpError.FLT_FLUVOLUM_TIME_PARA;		
					 iParaStep := 0;
		  ELSE
					rSetSpeed := stLocalPara.rFluVolumeSet * 60.0 / stRunPara.rSpeedRatio / stLocalPara.rRuntimeSet;
					IF rSetSpeed >= 0.001 AND  rSetSpeed <= 600 THEN
						iParaStep := iParaStep + 1;
					ELSE
						eERRORID := PumpError.FLT_FLUVOLUM_TIME_PARA;		
						iParaStep := 0;
			END_IF
		END_IF		
	2://读取液量（2word）、时间(2word)、间隔时间(2word)、灌装次数(word)、回吸角度(word)、运行方向(word)
			iOldParaStep:=iParaStep;
			wMBAddReadRegs:=1002;
			wQuantityReadRegs:=10;
			xReadRegs:=TRUE;
			IF  fbReadRegs.bBusy THEN
			 	xReadRegs:=FALSE;
				iParaStep:=iParaStep+1;
			END_IF
	3://等待读取完成
			 	iOldParaStep:=iParaStep;
	  	  IF  NOT 	fbReadRegs.bBusy AND  NOT  	fbReadRegs.bError THEN
				 				//液量
								stReadPara.rFluVolume:=M_Little_Endian(pInputData:=ADR(arwDataReadRegs[1]));
								//时间
								stReadPara.rRuntime:=M_Little_Endian(pInputData:=ADR(arwDataReadRegs[3]));
								
	  		 				 iParaStep:=iParaStep+1;
	  		 ELSIF   	fbReadRegs.bError THEN
	  		 			iParaStep:=999;				
	  		 			eErrorID:=PumpError.FLT_READ_PARA;					
	  		 END_IF	
	4://设定与显示进行比较
				iOldParaStep:=iParaStep;
				IF stLocalPara.rFluVolumeSet <> stReadPara.rFluVolume OR 
				 	 stLocalPara.rRuntimeSet <> stReadPara.rRuntime   THEN
					 iParaStep:=iParaStep + 1;	
				ELSE
					 iParaStep:=iParaStep+8;
				END_IF
	5://设定虚假时间
			 MEMCPY(ADR(arwSetData[1]),ADR(stLocalPara.rVirualTime),SIZEOF(stLocalPara.rVirualTime) ); 
			 arwDataWriteRegs[1]:=arwSetData[2];
			 arwDataWriteRegs[2]:=arwSetData[1];
			 iParaStep:=iParaStep +1;
	6://需要传送虚假的时间
			 iOldParaStep:=iParaStep;
			 wQuantityWriteRegs:=2;
			 wMBAddWriteRegs:=1004;
			 xWriteRegs:=TRUE;
			 IF  fbWriteRegs.bBusy THEN
					 xWriteRegs:=FALSE;
					 iParaStep:=iParaStep+1;
			END_IF	
	7://等待设定完成
				iOldParaStep:=iParaStep;
			 IF  NOT 	fbWriteRegs.bBusy AND  NOT  	fbWriteRegs.bError THEN
							  iParaStep:=iParaStep +1;
				ELSIF   	fbReadRegs.bError THEN
						 iParaStep:=999;				
						 eErrorID:=PumpError.FLT_SET_PARA;					
				END_IF				
  8://需要设定液量
			 iOldParaStep:=iParaStep;
			 MEMCPY(ADR(arwSetData[1]),ADR(stLocalPara.rFluVolumeSet),SIZEOF(stLocalPara.rFluVolumeSet) ); 
			 arwDataWriteRegs[1]:=arwSetData[2];
			 arwDataWriteRegs[2]:=arwSetData[1];
			 wQuantityWriteRegs:=2;
			 wMBAddWriteRegs:=1002;
			 xWriteRegs:=TRUE;
			 IF  fbWriteRegs.bBusy THEN
					 xWriteRegs:=FALSE;
					 iParaStep:=iParaStep+1;
			END_IF
	9://液量设定完成
			iOldParaStep:=iParaStep;
	  	IF  NOT 	fbWriteRegs.bBusy AND  NOT  	fbWriteRegs.bError THEN
	  	 				iParaStep:=iParaStep + 1;
	  	 ELSIF   	fbReadRegs.bError THEN
	  	 			iParaStep:=999;				
	  	 			eErrorID:=PumpError.FLT_SET_PARA;					
	  	 END_IF		
  10://设定运行时间
			 iOldParaStep:=iParaStep;
			 MEMCPY(ADR(arwSetData[1]),ADR(stLocalPara.rRuntimeSet),SIZEOF(stLocalPara.rRuntimeSet) ); 
			 arwDataWriteRegs[1]:=arwSetData[2];
			 arwDataWriteRegs[2]:=arwSetData[1];
			 wQuantityWriteRegs:=2;
			 wMBAddWriteRegs:=1004;
			 xWriteRegs:=TRUE;
			 IF  fbWriteRegs.bBusy THEN
					 xWriteRegs:=FALSE;
					 iParaStep:=iParaStep+1;
			END_IF
	11://等待时间设定完成
			iOldParaStep:=iParaStep;
	  	IF  NOT 	fbWriteRegs.bBusy AND  NOT  	fbWriteRegs.bError THEN
	  	 				iParaStep:=iParaStep + 1;
	  	 ELSIF   	fbReadRegs.bError THEN
	  	 			iParaStep:=999;				
	  	 			eErrorID:=PumpError.FLT_SET_PARA;					
	  	 END_IF		
	12://比较方向
				iOldParaStep:=iParaStep;
				stReadPara.iDirectionSet:=WORD_TO_INT(arwDataReadRegs[9]);
				IF stLocalPara.iDirectionSet<> stReadPara.iDirectionSet   THEN
										iParaStep:=iParaStep+1;	
				ELSE
										iParaStep:=iParaStep+3;	
				END_IF
	13://写入方向
			 iOldParaStep:=iParaStep;
			 MEMCPY(ADR(arwDataWriteRegs[1]),ADR(stLocalPara.iDirectionSet),SIZEOF (stLocalPara.iDirectionSet));
			 wQuantityWriteRegs:=1;
			 wMBAddWriteRegs:=1010;
			 xWriteRegs:=TRUE;
			 IF  fbWriteRegs.bBusy THEN
					 xWriteRegs:=FALSE;
					 iParaStep:=iParaStep+1;
			END_IF
  14://方向写入完成
			iOldParaStep:=iParaStep;
	  	IF  NOT 	fbWriteRegs.bBusy AND  NOT  	fbWriteRegs.bError THEN
	  	 				iParaStep:=iParaStep +1;
	  	 ELSIF   	fbReadRegs.bError THEN
	  	 			iParaStep:=999;				
	  	 			eErrorID:=PumpError.FLT_SET_PARA;					
	  	 END_IF		
	15://比较重复次数
				iOldParaStep:=iParaStep;
				//重复次数
				stReadPara.iCycleNumber:=WORD_TO_INT(arwDataReadRegs[7]);
				IF stLocalPara.iCycleNumber<> stReadPara.iCycleNumber   THEN
					 iParaStep:=iParaStep+1;	
				ELSE
					 iParaStep:=iParaStep+3;
				END_IF	
	16://写入重复次数
			 iOldParaStep:=iParaStep;
			 MEMCPY(ADR(arwDataWriteRegs[1]),ADR(stLocalPara.iCycleNumber),SIZEOF(stLocalPara.iCycleNumber));
			 wQuantityWriteRegs:=1;
			 wMBAddWriteRegs:=1008;
			 xWriteRegs:=TRUE;
			 IF  fbWriteRegs.bBusy THEN
					 xWriteRegs:=FALSE;
					 iParaStep:=iParaStep+1;
			END_IF
  17://重复次数写入完成
			iOldParaStep:=iParaStep;
	  	IF  NOT 	fbWriteRegs.bBusy AND  NOT  	fbWriteRegs.bError THEN
	  	 				iParaStep:=iParaStep +1;
	  	 ELSIF   	fbReadRegs.bError THEN
	  	 			iParaStep:=999;				
	  	 			eErrorID:=PumpError.FLT_SET_PARA;					
	  	 END_IF		
//////////////////////////待开放回吸角度/////////////////////////////////////////	 
	18://比较回吸角度
				iOldParaStep:=iParaStep;
				stReadPara.iBackAngle:=WORD_TO_INT(arwDataReadRegs[8]);
				IF stLocalPara.iBackAngle<> stReadPara.iBackAngle   THEN
					 iParaStep:=iParaStep+1;	
				ELSE
					 iParaStep:=iParaStep+3;
				END_IF	
	19://写入回吸角度
			 iOldParaStep:=iParaStep;
			 MEMCPY(ADR(arwDataWriteRegs[1]),ADR(stLocalPara.iBackAngle),SIZEOF(stLocalPara.iBackAngle));
			 wQuantityWriteRegs:=1;
			 wMBAddWriteRegs:=1009;
			 xWriteRegs:=TRUE;
			 IF  fbWriteRegs.bBusy THEN
					 xWriteRegs:=FALSE;
					 iParaStep:=iParaStep+1;
			END_IF
  20://写入回吸角度完成
			iOldParaStep:=iParaStep;
	  	IF  NOT 	fbWriteRegs.bBusy AND  NOT  	fbWriteRegs.bError THEN
	  	 				iParaStep:=iParaStep +1;
	  	 ELSIF   	fbReadRegs.bError THEN
	  	 			iParaStep:=999;				
	  	 			eErrorID:=PumpError.FLT_SET_PARA;					
	  	 END_IF				 
			 
	21://判断是否执行ModulePush
      IF   iOperType=stOperType.iModulePush THEN
						iParaStep:=iParaStep +1;
			ELSE
						iParaStep:=100;
			END_IF
	22://单元地址设定	
				 iOldParaStep:=iParaStep;
				 MEMCPY(ADR(arwDataWriteRegs[1]),ADR(stLocalPara.iModuleAdress),SIZEOF(stLocalPara.iModuleAdress));
				 wQuantityWriteRegs:=1;
				 wMBAddWriteRegs:=2000;
				 xWriteRegs:=TRUE;
				 IF  fbWriteRegs.bBusy THEN
						 xWriteRegs:=FALSE;
						 iParaStep:=iParaStep+1;
				END_IF
	23://单元地址设定完成
				iOldParaStep:=iParaStep;
				IF  NOT 	fbWriteRegs.bBusy AND  NOT  	fbWriteRegs.bError THEN
								iParaStep:=iParaStep +1;
				 ELSIF   	fbReadRegs.bError THEN
							iParaStep:=999;				
							eErrorID:=PumpError.FLT_SET_PARA;					
				 END_IF			
	24://写入回吸角度
				 iOldParaStep:=iParaStep;
				 MEMCPY(ADR(arwDataWriteRegs[1]),ADR(stLocalPara.iBackAngle),SIZEOF(stLocalPara.iBackAngle));
				 wQuantityWriteRegs:=1;
				 wMBAddWriteRegs:=1009;
				 xWriteRegs:=TRUE;
				 IF  fbWriteRegs.bBusy THEN
						 xWriteRegs:=FALSE;
						 iParaStep:=iParaStep+1;
				END_IF
	25://写入回吸角度完成
				iOldParaStep:=iParaStep;
				IF  NOT 	fbWriteRegs.bBusy AND  NOT  	fbWriteRegs.bError THEN
								iParaStep:=iParaStep +1;
				 ELSIF   	fbReadRegs.bError THEN
							iParaStep:=999;				
							eErrorID:=PumpError.FLT_SET_PARA;					
				 END_IF				 
	26://写入重复次数
			 iOldParaStep:=iParaStep;
			 MEMCPY(ADR(arwDataWriteRegs[1]),ADR(stLocalPara.iCycleNumber),SIZEOF(stLocalPara.iCycleNumber));
			 wQuantityWriteRegs:=1;
			 wMBAddWriteRegs:=1008;
			 xWriteRegs:=TRUE;
			 IF  fbWriteRegs.bBusy THEN
					 xWriteRegs:=FALSE;
					 iParaStep:=iParaStep+1;
			END_IF
  27://重复次数写入完成
			iOldParaStep:=iParaStep;
	  	IF  NOT 	fbWriteRegs.bBusy AND  NOT  	fbWriteRegs.bError THEN
	  	 				iParaStep:=100;
	  	 ELSIF   	fbReadRegs.bError THEN
	  	 			iParaStep:=999;				
	  	 			eErrorID:=PumpError.FLT_SET_PARA;					
	  	 END_IF				  

	//21://设定单元速度
	//		 iOldParaStep:=iParaStep;
	//		 MEMCPY(ADR(arwSetData[1]),ADR(stLocalPara.iModuleSpeed),SIZEOF(stLocalPara.iModuleSpeed) ); 
	//		 arwDataWriteRegs[1]:=arwSetData[2];
	//		 arwDataWriteRegs[2]:=arwSetData[1];
	//		 iParaStep:=iParaStep +1;
  //22://传送单元速度
	//		 iOldParaStep:=iParaStep;
	//		 wQuantityWriteRegs:=2;
	//		 wMBAddWriteRegs:=2001;
	//		 xWriteRegs:=TRUE;
	//		 IF  fbWriteRegs.bBusy THEN
	//				 xWriteRegs:=FALSE;
	//				 iParaStep:=iParaStep+1;
	//		END_IF	
	//23://等待设定完成
	//			iOldParaStep:=iParaStep;
	//		 IF  NOT 	fbWriteRegs.bBusy AND  NOT  	fbWriteRegs.bError THEN
	//						  iParaStep:=100;
	//			ELSIF   	fbReadRegs.bError THEN
	//					 iParaStep:=999;				
	//					 eErrorID:=PumpError.FLT_SET_PARA;					
	//			END_IF				
	100://参数写入完成
				iOperType:=stOperType.iWait;
				stPara.xBusy:=FALSE;
				stPara.xDone:=TRUE;
				iParaStep:=0;		
	ELSE
		;	
END_CASE
//防止程序二次执行
IF   stPara.xBusy THEN
		 stPara.xStart:=FALSE;
END_IF
END_ACTION

END_FUNCTION_BLOCK

(* stored: Version 1.1.0.1, ProductVersion 3.1.4024.9
   POU FB_KF300: Id {d17c1c4b-fe6d-4914-b0e5-26831df67b43}, SpecialFunc None
   Action ACT_Calibration: Id {e04bb569-1c60-418c-908e-e90a0e6ac504}
   Action ACT_Error: Id {8e071d61-e5ef-43ab-8951-287a6ba9ed2b}
   Action ACT_Operation: Id {69bd1712-87b9-4687-a4b7-427e7b5c2cee}
   Action ACT_ParaCalc: Id {082b3045-a19d-4f59-a04c-cbfd47d9616e}
   Action ACT_Reset: Id {eb57277f-057a-445d-b2fc-44fbe77c82fc}
   Action ACT_Running: Id {f72b25a7-4f66-439b-b942-35021509e771}
   Action ACT_RunPara: Id {de4ccdf8-7874-4800-9b27-4ec05af2e4ab} *)
